(* PLC project Unnamed, Unknown Unnamed 1 *)
(* stored: creationDateTime 2022-12-09T12:13:26, modificationDateTime 2022-12-16T11:30:15 *)

PROGRAM program0
  VAR
    CSV_NAME_0 : HMI_STRING := 'my_int_csv.csv';
    CSV_NAME_1 : HMI_STRING := 'my_str_csv.csv';
    CSV_ROWSTR : HMI_STRING := 'Recipe 5';
    CSV_COLSTR : HMI_STRING := 'Ingredient D';
    CSV_ROWIDX : HMI_INT := 5;
    CSV_COLIDX : HMI_INT := 4;
    csv_read_by_string0 : csv_read_by_string;
    csv_read_by_int0 : csv_read_by_int;
    csv_reload0 : csv_reload;
    CSV_RES_0 : HMI_STRING;
    CSV_RES_1 : HMI_STRING;
    CSV_ACK_0 : HMI_BOOL;
    CSV_ACK_1 : HMI_BOOL;
    CSV_RELOAD_BTN : HMI_BOOL;
  END_VAR

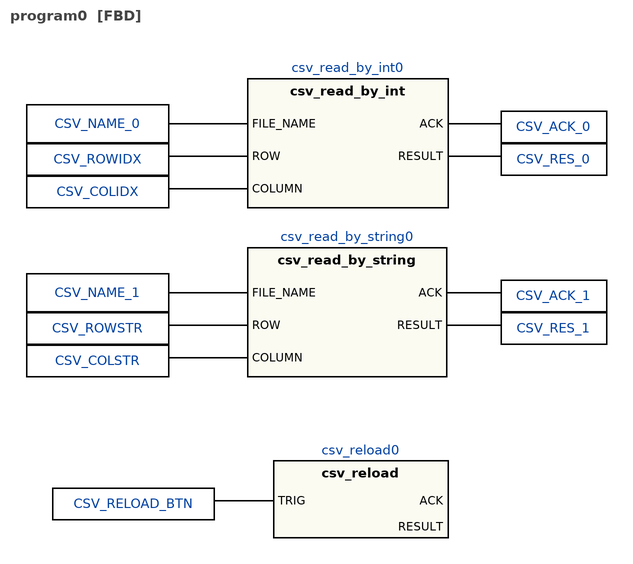
(* FBD diagram, written out as Structured Text *)
csv_read_by_int0(FILE_NAME := CSV_NAME_0, ROW := CSV_ROWIDX, COLUMN := CSV_COLIDX);
CSV_ACK_0 := csv_read_by_int0.ACK;
CSV_RES_0 := csv_read_by_int0.RESULT;
csv_read_by_string0(FILE_NAME := CSV_NAME_1, ROW := CSV_ROWSTR, COLUMN := CSV_COLSTR);
CSV_ACK_1 := csv_read_by_string0.ACK;
CSV_RES_1 := csv_read_by_string0.RESULT;
csv_reload0(TRIG := CSV_RELOAD_BTN);
END_PROGRAM

CONFIGURATION config
  RESOURCE resource1 ON PLC
    TASK task0(INTERVAL := T#20ms, PRIORITY := 0);
    PROGRAM instance0 WITH task0 : program0;
  END_RESOURCE
END_CONFIGURATION
